Universal Robots PolyScope program: network_comm.urp

Program network_comm (installation=default directory=/programs/usbdisk/new folder/new folder_1 createdIn=5.8.0.10253 lastSavedIn=5.8.0.10253 robotSerialNumber=20205501115)
Calibrated DH parameters: a=[0.000276, -0.406003, -0.392048, 0.000048, 0.00004, 0]; d=[0.162697, -327.101782, 328.941291, -1.70618, 0.099534, 0.099542]; alpha=[1.570908, -0.000386, 0.008812, 1.568492, -1.569726, 0]; deltaTheta=[0, 0.301365, 6.023141, -0.041322, 0, 0]
BeforeStart
  Popup Message (haltProgram=false message=Ok to open gripper? inputType=Text)
  URCap Gripper Activate (Robotiq_Grippers, Robotiq Inc.) dataModel(ResetAndActivateKey=false)
  URCap Gripper (Robotiq_Grippers, Robotiq Inc.) dataModel(position=100.0, force=0.0, speed=0.0, positionInDouble=100.0, forceInDouble=0.0, speedInDouble=0.0, slaveIds=[9], blocking=true)
  Script: socket_close("robot_socket")
  Wait Sleep waitTime=2
  Script: socket_open("172.31.1.96", 30000, "robot_socket")
  task := [0,0]
  receive_data := [6, 0, 0, 0, 0, 0, 0]
  transmit_data := [0, 0, 0, 0, 0, 0]
  move_to_joints := [d2r(90), d2r(-90), d2r(60), d2r(300), d2r(-90), d2r(-180)]
  SuppressedNode
    Call Init_joint
  move_to_tcp := get_target_tcp_pose()
  is_tcp_rec := False
  is_joint_rec := False
  is_tcp_send := False
  is_joint_send := False
Robot Program (runOnlyOnce=false)
  Wait Sleep waitTime=2
  task := socket_read_ascii_float(1, "robot_socket")
  Switch expression=task[1]
    Case (caseValue=1)
      is_joint_rec := True
      Call Receive_msg
    Case (caseValue=2)
      is_joint_send := True
      Call Transmit_msg
    Case (caseValue=3)
      Call OpenGripper
    Case (caseValue=4)
      Call CloseGripper
    Case (caseValue=5)
      is_tcp_send := True
      Call Transmit_msg
    Case (caseValue=6)
      is_tcp_rec := True
      Call Receive_msg
SuppressedNode
  SubProgram -> Init_joint
SubProgram -> Receive_msg
SubProgram -> Transmit_msg
SubProgram -> OpenGripper
SubProgram -> CloseGripper
Thread Thread_1 (runOnlyOnce=false)
  If is_tcp_rec
    Script: movel(move_to_tcp, a=0.1, v=0.15, r=0)
    is_tcp_rec := False
  ElseIf is_joint_rec
    Script: movej(move_to_joints, a=0.1, v=0.15, t=0, r=0)
    is_joint_rec := False
  Wait Sleep waitTime=1
SubProgram Init_joint (keepSynchronizedWithDisk=false)
  If get_actual_joint_positions()≠move_to_joints
    Script: movej(move_to_joints, a=0.1, v=0.15, t=0, r=0)
    Wait Sleep waitTime=2
SubProgram Receive_msg (keepSynchronizedWithDisk=false)
  receive_data := socket_read_ascii_float(6, "robot_socket")
  If receive_data[0]≠6
    Script: socket_send_string("0", "robot_socket")
  Else 
    Script: socket_send_string("1", "robot_socket")
    i := 0
    If is_tcp_rec
      Loop While (checkContinuously=false) expression=i<receive_data[0]
        Script: move_to_tcp[i] = receive_data[i+1]
        i := i+1
    ElseIf is_joint_rec
      Loop While (checkContinuously=false) expression=i<receive_data[0]
        Script: move_to_joints[i] = receive_data[i+1]
        i := i+1
  task := [0,0]
SubProgram Transmit_msg (keepSynchronizedWithDisk=false)
  If is_tcp_send
    curr_tcp_pose := get_actual_tcp_pose()
    i := 0
    Loop While (checkContinuously=false) expression=i<length(transmit_data)
      Script: transmit_data[i] = curr_tcp_pose[i]
      i := i+1
    is_tcp_send := False
  ElseIf is_joint_send
    transmit_data := get_actual_joint_positions()
    is_joint_send := False
  Script: socket_send_string(transmit_data,  "robot_socket")
  task := [0,0]
SubProgram OpenGripper (keepSynchronizedWithDisk=false)
  URCap Gripper (Robotiq_Grippers, Robotiq Inc.) dataModel(position=0.0, force=100.0, speed=100.0, positionInDouble=0.0, forceInDouble=100.0, speedInDouble=100.0, slaveIds=[9], blocking=true)
  Wait Sleep waitTime=0.01
  Script: socket_send_string("1", "robot_socket")
  task := [0,0]
SubProgram CloseGripper (keepSynchronizedWithDisk=false)
  URCap Gripper (Robotiq_Grippers, Robotiq Inc.) dataModel(position=100.0, force=100.0, speed=100.0, positionInDouble=100.0, forceInDouble=100.0, speedInDouble=100.0, slaveIds=[9], blocking=true)
  Wait Sleep waitTime=0.01
  Script: socket_send_string("1", "robot_socket")
  task := [0,0]
